// TwinCAT 3 PLC project CCS
// ProgramVersion: 3.1.4022.3
// libraries:
//   Tc2_Standard, * (Beckhoff Automation GmbH)
//   Tc2_System, * (Beckhoff Automation GmbH)
//   Tc3_EventLogger, * (Beckhoff Automation GmbH)
//   Tc3_Module, * (Beckhoff Automation GmbH)
// project tree:
//   DUTs/ AxisStatus.TcDUT, ChangeAxisEnable.TcDUT, ChangeOutputLine.TcDUT, ClearAllFaults.TcDUT, ClearAxisFaults.TcDUT, ControllerStatus.TcDUT, DisableAllAxes.TcDUT, EnableAllAxes.TcDUT, HomeAxis.TcDUT, IncomingMessage.TcDUT, IOStatus.TcDUT, MessageID.TcDUT, MoveAxisAbsolute.TcDUT, MoveAxisRelative.TcDUT, OutgoingMessage.TcDUT, StopAllMotion.TcDUT
//   GVLs/ CT.TcGVL, MSG.TcGVL
//   / PlcTask.TcTTO
//   POUs/ MAIN.TcPOU, newMessage.TcPOU, printChangeAxisEnable.TcPOU

CONFIGURATION CCS
    RESOURCE PLC ON TwinCAT3
        TASK PlcTask(INTERVAL := T#10ms, PRIORITY := 20);
        PROGRAM MAIN WITH PlcTask : MAIN;
    END_RESOURCE
END_CONFIGURATION

// ---- DUTs/AxisStatus.TcDUT
{attribute 'pack_mode' := '1'}
TYPE AxisStatus EXTENDS OutgoingMessage :
STRUCT
	axisIndex: INT; (* 1 or 2. *)
	enabled: BOOL; (* Axis enabled? *)
	moving: BOOL;  (* Axis moving? *)
	atHome: BOOL;   (* Axis has been homed? *)
	atLowLimit: BOOL; (* Axis at low limit switch? *)
	atHighLimit: BOOL; (* Axis at high limit switch? *)
	errorCode: DINT;
	position: LREAL;
END_STRUCT
END_TYPE

// ---- DUTs/ChangeAxisEnable.TcDUT
{attribute 'pack_mode' := '1'}
TYPE ChangeAxisEnable EXTENDS IncomingMessage :
STRUCT
	axisIndex: INT; (* 1 or 2.*)
	enabled: BOOL;
END_STRUCT
END_TYPE

// ---- DUTs/ChangeOutputLine.TcDUT
{attribute 'pack_mode' := '1'}
TYPE ChangeOutputLine EXTENDS IncomingMessage :
STRUCT
	lineIndex: DINT;
	newState: BOOL;
END_STRUCT
END_TYPE

// ---- DUTs/ClearAllFaults.TcDUT
{attribute 'pack_mode' := '1'}
TYPE ClearAllFaults EXTENDS IncomingMessage :
STRUCT
END_STRUCT
END_TYPE

// ---- DUTs/ClearAxisFaults.TcDUT
{attribute 'pack_mode' := '1'}
TYPE ClearAxisFaults EXTENDS IncomingMessage :
STRUCT
	axisIndex: INT; (* 1 or 2.*)
END_STRUCT
END_TYPE

// ---- DUTs/ControllerStatus.TcDUT
{attribute 'pack_mode' := '1'}
TYPE ControllerStatus EXTENDS OutgoingMessage :
STRUCT
	commLinkStatus: STRING(CT.STATUS_STRING_SIZE);
	motionEnabled: BOOL;
	lastCommandStatus: STRING(CT.STATUS_STRING_SIZE);
END_STRUCT
END_TYPE

// ---- DUTs/DisableAllAxes.TcDUT
{attribute 'pack_mode' := '1'}
TYPE DisableAllAxes EXTENDS IncomingMessage :
STRUCT
END_STRUCT
END_TYPE

// ---- DUTs/EnableAllAxes.TcDUT
{attribute 'pack_mode' := '1'}
TYPE EnableAllAxes EXTENDS IncomingMessage :
STRUCT
END_STRUCT
END_TYPE

// ---- DUTs/HomeAxis.TcDUT
{attribute 'pack_mode' := '1'}
TYPE HomeAxis EXTENDS IncomingMessage :
STRUCT
	axisIndex: INT; (* 1 or 2.*)
END_STRUCT
END_TYPE

// ---- DUTs/IncomingMessage.TcDUT
{attribute 'pack_mode' := '1'}
TYPE IncomingMessage :
STRUCT
	id: MessageID;   (* Used to identify new messages. *)
	version: LINT;   (* Matches serialVersionUID of the equivalent Java class. *)
END_STRUCT
END_TYPE

// ---- DUTs/IOStatus.TcDUT
{attribute 'pack_mode' := '1'}
TYPE IOStatus EXTENDS OutgoingMessage :
STRUCT
	digitalInputs: DINT;  (* Bit mask of current states. *)
	digitalOutputs: DINT; (* Bit mask of current states. *)
	analogInputs: ARRAY [0..CT.ANALOG_ARRAY_SIZE-1] OF LREAL; (* Current analog readings. *)
END_STRUCT
END_TYPE

// ---- DUTs/MessageID.TcDUT
{attribute 'pack_mode' := '1'}
(* At least one of these components must change for each new
   message sent. 
 *)
TYPE MessageID :
STRUCT
	ipv4: DINT;       (* IP address of sender. *)
	pid: DINT;        (* Sender process ID. *)
	dtime: DINT;      (* Time of day in milliseconds. *)
	sequence: DINT;   (* Message sequence number. *)
END_STRUCT
END_TYPE

// ---- DUTs/MoveAxisAbsolute.TcDUT
{attribute 'pack_mode' := '1'}
TYPE MoveAxisAbsolute EXTENDS IncomingMessage :
STRUCT
	axisIndex: INT; (* 1 or 2.*)
	position: LREAL;
	speed: LREAL;
END_STRUCT
END_TYPE

// ---- DUTs/MoveAxisRelative.TcDUT
{attribute 'pack_mode' := '1'}
TYPE MoveAxisRelative EXTENDS IncomingMessage :
STRUCT
	axisIndex: INT; (* 1 or 2.*)
	distance: LREAL;
	moveTime: TIME;
END_STRUCT
END_TYPE

// ---- DUTs/OutgoingMessage.TcDUT
{attribute 'pack_mode' := '1'}
TYPE OutgoingMessage :
STRUCT
	version: LINT; (* Matches the serialVersionUID of the equivalent Java class.*)
END_STRUCT
END_TYPE

// ---- DUTs/StopAllMotion.TcDUT
{attribute 'pack_mode' := '1'}
TYPE StopAllMotion EXTENDS IncomingMessage :
STRUCT
END_STRUCT
END_TYPE

// ---- GVLs/CT.TcGVL
{attribute 'qualified_only'}
VAR_GLOBAL CONSTANT
	AXIS_NAME_SIZE: DINT := 9;
	FAULT_STRING_SIZE: DINT := 19;
	FAULT_ARRAY_SIZE: DINT := 10;
	STATUS_STRING_SIZE: DINT := 19;
	ANALOG_ARRAY_SIZE : DINT := 20;
END_VAR

// ---- GVLs/MSG.TcGVL
{attribute 'qualified_only'}
VAR_GLOBAL
	changeAxisEnable: FB_TcMessage;
END_VAR

// ---- POUs/MAIN.TcPOU
PROGRAM MAIN
VAR
	(* Messages sent to CCS. *)
	outAxisStatus: AxisStatus;
	outControllerStatus: ControllerStatus;
	outIOStatus: IOStatus;
	ackChangeAxisEnable: ChangeAxisEnable;
	ackChangeOutputLine: ChangeOutputLine;
	ackClearAllFaults: ClearAllFaults;
	ackClearAxisFaults: ClearAxisFaults;
	ackEnableAllAxes: EnableAllAxes;
	ackDisableAllAxes: DisableAllAxes;
	ackMoveAxisRelative: MoveAxisRelative;
	ackMoveAxisAbsolute: MoveAxisAbsolute;
	ackHomeAxis: HomeAxis;
	
	(* Messages coming from CCS. *)
	inChangeAxisEnable: ChangeAxisEnable;
	inChangeOutputLine: ChangeOutputLine;
	inClearAllFaults: ClearAllFaults;
	inClearAxisFaults: ClearAxisFaults;
	inEnableAllAxes: EnableAllAxes;
	inDisableAllAxes: DisableAllAxes;
	inMoveAxisRelative: MoveAxisRelative;
	inMoveAxisAbsolute: MoveAxisAbsolute;
	inHomeAxis: HomeAxis;

	firstCycle: BOOL := TRUE;
END_VAR

VAR CONSTANT
	zeroID: MessageID := (ipv4 := 0, pid := 0, dtime := 0, sequence := 0);
END_VAR

(* Initialization. *)
IF firstCycle THEN
	firstCycle := FALSE;
	ackChangeAxisEnable.id := inChangeAxisEnable.id := zeroID;
	ackChangeOutputLine.id := inChangeOutputLine.id := zeroID;
	ackClearAllFaults.id := inClearAllFaults.id := zeroID;
	ackClearAxisFaults.id := inClearAxisFaults.id := zeroID;
	ackEnableAllAxes.id := inEnableAllAxes.id := zeroID;
	ackDisableAllAxes.id := inDisableAllAxes.id := zeroID;
	ackMoveAxisRelative.id := inMoveAxisRelative.id := zeroID;
	ackMoveAxisAbsolute.id := inMoveAxisAbsolute.id := zeroID;
	ackHomeAxis.id := inHomeAxis.id := zeroID;
	
	MSG.changeAxisEnable.CreateEx(ST_ShutterEvent.ChangeAxisEnable, 0);
END_IF

(* Check for arrival of new messages. *)
IF newMessage(inChangeAxisEnable, ackChangeAxisEnable) THEN
	ackChangeAxisEnable := inChangeAxisEnable;
	printChangeAxisEnable(ackChangeAxisEnable);
END_IF

END_PROGRAM

// ---- POUs/newMessage.TcPOU
FUNCTION newMessage : BOOL
VAR_INPUT
	first: IncomingMessage;
	second: IncomingMessage;
END_VAR
VAR
END_VAR

newMessage := (first.id.dtime <> second.id.dtime)
	OR (first.id.ipv4 <> second.id.ipv4)
	OR (first.id.pid <> second.id.pid)
    OR (first.id.sequence <> second.id.sequence);

END_FUNCTION

// ---- POUs/printChangeAxisEnable.TcPOU
FUNCTION printChangeAxisEnable : BOOL
VAR_INPUT
	cmd: ChangeAxisEnable;
END_VAR
VAR
END_VAR

MSG.changeAxisEnable.ipArguments.Clear().AddInt(cmd.axisIndex).AddBool(cmd.enabled);
MSG.changeAxisEnable.Send(0);

END_FUNCTION
